SUBAPPLICATION Softkey_Aux_Web_IXA (* VT-SoftKey lesen ODER AUX-Zuweisung (Joystick) lesen ODER lokaler Web-Override (z.B. vt-ui-mirror auf demselben Modul) -> 1 gemeinsamer, kontinuierlicher AX-Pegel (kein Remote-Write, kein Event) - fuer Tastbetrieb (Jog/Tippen), bei dem der Pegel selbst (nicht eine Flanke) weiterverarbeitet werden soll, z.B. als G-Eingang eines AX_AX_SEL_AR oder als DI1 einer GreenWhiteBackground-Ruecklmeldung. Kommando-Haelfte von Softkey_Aux_IXA_TO_Remote_WRITE, aber OUT statt Remote-Write. *)
  (* Standard: 61499-2; Description: Copyright (c) 2026 Meisterschulen am Ostbahnhof This program and the accompanying materials are made available under the terms of the Eclipse Public License 2.0 which is available at https://www.eclipse.org/legal/epl-2.0/ SPDX-License-Identifier: EPL-2.0 *)
  (* Version 1.0, 2026-09-13, Franz Höpfinger, Meisterschulen am Ostbahnhof, initial implementation - herausgeloest aus Softkey_Aux_IXA_TO_Remote_WRITE (Quellen-ODER ohne den Remote-Write-Teil), fuer Bunkerboden (2 tastende Kommandos, Max/Wert, die lokal zu einem PWM-Prozentwert selektiert werden muessen statt direkt remote geschrieben zu werden). *)
  PACKAGE MyLib::sys;
  IMPORT isobus::UT::Q::const::IDs::ID_NULL;
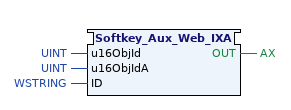
  VAR_INPUT
    u16ObjId : UINT := ID_NULL; (* Object ID SoftKey (VT) *)
    u16ObjIdA : UINT := ID_NULL; (* Object ID AuxFunction2 (VT) *)
    ID : WSTRING; (* Lokale Subscribe-Adresse fuer einen Web-Client (z.B. vt-ui-mirror) auf demselben Modul, ODER-verknuepft mit SoftKey und AUX *)
  END_VAR
  PLUGS
    OUT : adapter::types::unidirectional::AX; (* SoftKey ODER Aux ODER Web-Override, kontinuierlicher Pegel (TRUE solange gehalten/aktiv) *)
  END_PLUGS
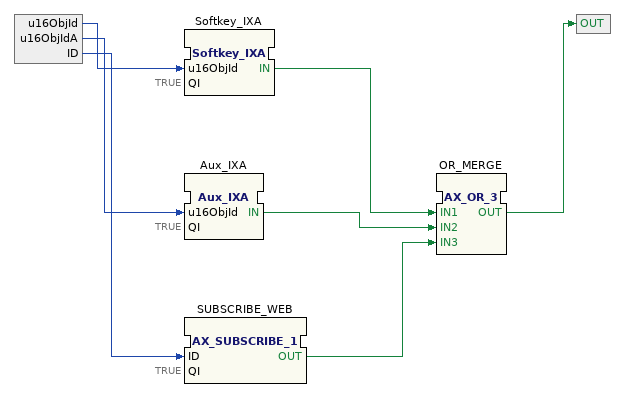
  FBS
    Softkey_IXA : isobus::UT::io::Softkey::Softkey_IXA(QI := TRUE);
    Aux_IXA : isobus::UT::io::Auxiliary::IN::Aux_IXA(QI := TRUE);
    SUBSCRIBE_WEB : adapter::net::AX_SUBSCRIBE_1(QI := TRUE);
    OR_MERGE : adapter::booleanOperators::AX_OR_3;
  END_FBS
  DATA_CONNECTIONS
    u16ObjId TO Softkey_IXA.u16ObjId;
    u16ObjIdA TO Aux_IXA.u16ObjId;
    ID TO SUBSCRIBE_WEB.ID;
  END_CONNECTIONS
  ADAPTER_CONNECTIONS
    Softkey_IXA.IN TO OR_MERGE.IN1;
    Aux_IXA.IN TO OR_MERGE.IN2;
    SUBSCRIBE_WEB.OUT TO OR_MERGE.IN3;
    OR_MERGE.OUT TO OUT;
  END_CONNECTIONS
END_SUBAPPLICATION
